PROGRAM P_Outputs
VAR
END_VAR

///////////////////// Lights //////////////////////////////

IF G_Inputs.bRedButton THEN 
	G_Outputs.bRedButtonLight := FALSE;
ELSE 
	G_Outputs.bRedButtonLight := TRUE;
END_IF

IF G_Inputs.bGreenButton THEN 
	G_Outputs.bGreenButtonLight := TRUE;
ELSE 
	G_Outputs.bGreenButtonLight := FALSE;
END_IF


IF G_Inputs.bManualModeSelector OR G_Inputs.bAutoModeSelector THEN
	G_Outputs.bGreenButtonLight := FALSE;
	G_Outputs.bRedButtonLight := TRUE;
ELSE
	G_Outputs.bGreenButtonLight := TRUE;
	G_Outputs.bRedButtonLight := FALSE;
END_IF

END_PROGRAM

(* stored: Version 1.1.0.1, ProductVersion 3.1.4024.12
   POU P_Outputs: Id {05725e2c-789e-4faf-9ddc-3f7ec72a2093}, SpecialFunc None *)
